LIN {X 0,Y 72.72,Z 376.859,A -85,B 0,C 180,E1 -30203.104,E2 -30203.104} C_VEL
LIN {X 0,Y 74.834,Z 373.573,A -85,B 0,C 180,E1 -30209.448,E2 -30209.448} C_VEL
LIN {X 0,Y 76.166,Z 370.91,A -85,B 0,C 180,E1 -30214.53,E2 -30214.53} C_VEL
LIN {X 0,Y 77.498,Z 367.967,A -85,B 0,C 180,E1 -30221.527,E2 -30221.527} C_VEL
LIN {X 0,Y 78.253,Z 365.544,A -85,B 0,C 180,E1 -30229.683,E2 -30229.683} C_VEL
LIN {X 0,Y 78.687,Z 364.699,A -85,B 0,C 180,E1 -30234.216,E2 -30234.216} C_VEL
LIN {X 0,Y 78.512,Z 364.725,A -85,B 0,C 180,E1 -30236.541,E2 -30236.541} C_VEL
LIN {X 0,Y 77.196,Z 365.763,A -85,B 0,C 180,E1 -30239.68,E2 -30239.68} C_VEL
LIN {X 0,Y 72.784,Z 369.848,A -85,B 0,C 180,E1 -30247.513,E2 -30247.513} C_VEL
LIN {X 0,Y 72.396,Z 370.336,A -85,B 0,C 180,E1 -30249.099,E2 -30249.099} C_VEL
LIN {X 0,Y 71.855,Z 371.227,A -85,B 0,C 180,E1 -30252.026,E2 -30252.026} C_VEL
LIN {X 0,Y 71.087,Z 372.22,A -85,B 0,C 180,E1 -30254.34,E2 -30254.34} C_VEL
LIN {X 0,Y 69.527,Z 373.648,A -85,B 0,C 180,E1 -30256.205,E2 -30256.205} C_VEL
LIN {X 0,Y 68.06,Z 374.817,A -85,B 0,C 180,E1 -30257.224,E2 -30257.224} C_VEL
LIN {X 0,Y 57.01,Z 381.349,A -85,B 0,C 180,E1 -30262.4,E2 -30262.4} C_VEL
LIN {X 0,Y 47.981,Z 385.676,A -85,B 0,C 180,E1 -30268.5,E2 -30268.5} C_VEL
LIN {X 0,Y 42.377,Z 388.048,A -85,B 0,C 180,E1 -30273.983,E2 -30273.983} C_VEL
LIN {X 0,Y 37.23,Z 389.851,A -85,B 0,C 180,E1 -30280.969,E2 -30280.969} C_VEL
LIN {X 0,Y 29.547,Z 392.319,A -85,B 0,C 180,E1 -30301.595,E2 -30301.595} C_VEL
LIN {X 0,Y 27.527,Z 392.919,A -85,B 0,C 180,E1 -30315.208,E2 -30315.208} C_VEL
LIN {X 0,Y 27.087,Z 393.084,A -85,B 0,C 180,E1 -30330,E2 -30330} C_VEL
LIN {X 0,Y 27.51,Z 392.918,A -85,B 0,C 180,E1 -30344.801,E2 -30344.801} C_VEL
LIN {X 0,Y 29.494,Z 392.317,A -85,B 0,C 180,E1 -30358.461,E2 -30358.461} C_VEL
LIN {X 0,Y 37.219,Z 389.851,A -85,B 0,C 180,E1 -30379.051,E2 -30379.051} C_VEL
LIN {X 0,Y 45.142,Z 386.896,A -85,B 0,C 180,E1 -30388.898,E2 -30388.898} C_VEL
LIN {X 0,Y 53.964,Z 382.905,A -85,B 0,C 180,E1 -30395.73,E2 -30395.73} C_VEL
LIN {X 0,Y 63.273,Z 377.774,A -85,B 0,C 180,E1 -30400.743,E2 -30400.743} C_VEL
LIN {X 0,Y 68.055,Z 374.817,A -85,B 0,C 180,E1 -30402.789,E2 -30402.789} C_VEL
LIN {X 0,Y 69.524,Z 373.648,A -85,B 0,C 180,E1 -30403.803,E2 -30403.803} C_VEL
LIN {X 0,Y 71.069,Z 372.231,A -85,B 0,C 180,E1 -30405.656,E2 -30405.656} C_VEL
LIN {X 0,Y 72.083,Z 370.933,A -85,B 0,C 180,E1 -30408.723,E2 -30408.723} C_VEL
LIN {X 0,Y 73.11,Z 369.368,A -85,B 0,C 180,E1 -30414.452,E2 -30414.452} C_VEL
LIN {X 0,Y 73.872,Z 368.359,A -85,B 0,C 180,E1 -30419.968,E2 -30419.968} C_VEL
LIN {X 0,Y 72.867,Z 369.184,A -85,B 0,C 180,E1 -30426.331,E2 -30426.331} C_VEL
LIN {X 0,Y 72.009,Z 370.387,A -85,B 0,C 180,E1 -30432.587,E2 -30432.587} C_VEL
LIN {X 0,Y 71.53,Z 371.492,A -85,B 0,C 180,E1 -30437.108,E2 -30437.108} C_VEL
LIN {X 0,Y 70.166,Z 373.929,A -85,B 0,C 180,E1 -30443.581,E2 -30443.581} C_VEL
LIN {X 0,Y 69.095,Z 375.402,A -85,B 0,C 180,E1 -30447.196,E2 -30447.196} C_VEL
LIN {X 0,Y 67.095,Z 378.1,A -85,B 0,C 180,E1 -30453.075,E2 -30453.075} C_VEL
LIN {X 0,Y 63.076,Z 382.804,A -85,B 0,C 180,E1 -30464.263,E2 -30464.263} C_VEL
LIN {X 0,Y 61.501,Z 386.014,A -85,B 0,C 180,E1 -30475.155,E2 -30475.155} C_VEL
LIN {X 0,Y 62.216,Z 387.991,A -85,B 0,C 180,E1 -30484.551,E2 -30484.551} C_VEL
LIN {X 0,Y 66.715,Z 389.818,A -85,B 0,C 180,E1 -30497.838,E2 -30497.838} C_VEL
LIN {X 0,Y 70.841,Z 390.257,A -85,B 0,C 180,E1 -30504.307,E2 -30504.307} C_VEL
LIN {X 0,Y 75.986,Z 390.258,A -85,B 0,C 180,E1 -30510,E2 -30510} C_VEL
LIN {X 0,Y 70.616,Z 390.238,A -85,B 0,C 180,E1 -30515.961,E2 -30515.961} C_VEL
LIN {X 0,Y 65.397,Z 389.543,A -85,B 0,C 180,E1 -30524.869,E2 -30524.869} C_VEL
LIN {X 0,Y 61.939,Z 387.669,A -85,B 0,C 180,E1 -30536.991,E2 -30536.991} C_VEL
LIN {X 0,Y 61.564,Z 385.453,A -85,B 0,C 180,E1 -30547.024,E2 -30547.024} C_VEL
LIN {X 0,Y 63.998,Z 381.588,A -85,B 0,C 180,E1 -30558.837,E2 -30558.837} C_VEL
LIN {X 0,Y 67.094,Z 378.1,A -85,B 0,C 180,E1 -30566.926,E2 -30566.926} C_VEL
LIN {X 0,Y 69.778,Z 374.487,A -85,B 0,C 180,E1 -30575.019,E2 -30575.019} C_VEL
LIN {X 0,Y 70.905,Z 372.605,A -85,B 0,C 180,E1 -30579.738,E2 -30579.738} C_VEL
LIN {X 0,Y 71.576,Z 371.46,A -85,B 0,C 180,E1 -30582.904,E2 -30582.904} C_VEL
LIN {X 0,Y 72.257,Z 370.036,A -85,B 0,C 180,E1 -30588.817,E2 -30588.817} C_VEL
LIN {X 0,Y 73.07,Z 368.988,A -85,B 0,C 180,E1 -30594.822,E2 -30594.822} C_VEL
LIN {X 0,Y 73.883,Z 368.35,A -85,B 0,C 180,E1 -30600.032,E2 -30600.032} C_VEL
LIN {X 0,Y 73.103,Z 369.373,A -85,B 0,C 180,E1 -30605.549,E2 -30605.549} C_VEL
LIN {X 0,Y 72.396,Z 370.336,A -85,B 0,C 180,E1 -30609.099,E2 -30609.099} C_VEL
LIN {X 0,Y 71.537,Z 371.196,A -85,B 0,C 180,E1 -30610.75,E2 -30610.75} C_VEL
LIN {X 0,Y 69.503,Z 372.798,A -85,B 0,C 180,E1 -30612.197,E2 -30612.197} C_VEL
LIN {X 0,Y 65.793,Z 375.28,A -85,B 0,C 180,E1 -30613.316,E2 -30613.316} C_VEL
LIN {X 0,Y 56.47,Z 380.309,A -85,B 0,C 180,E1 -30614.749,E2 -30614.749} C_VEL
LIN {X 0,Y 55.18,Z 380.901,A -85,B 0,C 180,E1 -30615.229,E2 -30615.229} C_VEL
LIN {X 0,Y 45.014,Z 385.481,A -85,B 0,C 180,E1 -30620.486,E2 -30620.486} C_VEL
LIN {X 0,Y 38.846,Z 387.852,A -85,B 0,C 180,E1 -30625.233,E2 -30625.233} C_VEL
LIN {X 0,Y 32.995,Z 389.656,A -85,B 0,C 180,E1 -30631.571,E2 -30631.571} C_VEL
LIN {X 0,Y 23.526,Z 392.123,A -85,B 0,C 180,E1 -30653.313,E2 -30653.313} C_VEL
LIN {X 0,Y 20.721,Z 392.724,A -85,B 0,C 180,E1 -30670.174,E2 -30670.174} C_VEL
LIN {X 0,Y 19.994,Z 392.889,A -85,B 0,C 180,E1 -30690,E2 -30690} C_VEL
LIN {X 0,Y 20.704,Z 392.723,A -85,B 0,C 180,E1 -30709.843,E2 -30709.843} C_VEL
LIN {X 0,Y 23.483,Z 392.122,A -85,B 0,C 180,E1 -30726.765,E2 -30726.765} C_VEL
LIN {X 0,Y 32.987,Z 389.655,A -85,B 0,C 180,E1 -30748.45,E2 -30748.45} C_VEL
LIN {X 0,Y 41.907,Z 386.701,A -85,B 0,C 180,E1 -30757.271,E2 -30757.271} C_VEL
LIN {X 0,Y 51.45,Z 382.71,A -85,B 0,C 180,E1 -30762.974,E2 -30762.974} C_VEL
LIN {X 0,Y 61.285,Z 377.577,A -85,B 0,C 180,E1 -30767.077,E2 -30767.077} C_VEL
LIN {X 0,Y 64.617,Z 375.658,A -85,B 0,C 180,E1 -30768.196,E2 -30768.196} C_VEL
LIN {X 0,Y 66.311,Z 374.202,A -85,B 0,C 180,E1 -30771.201,E2 -30771.201} C_VEL
LIN {X 0,Y 66.824,Z 373.516,A -85,B 0,C 180,E1 -30773.928,E2 -30773.928} C_VEL
LIN {X 0,Y 67.857,Z 372.402,A -85,B 0,C 180,E1 -30779.965,E2 -30779.965} C_VEL
LIN {X 0,Y 66.889,Z 373.083,A -85,B 0,C 180,E1 -30785.995,E2 -30785.995} C_VEL
LIN {X 0,Y 65.56,Z 374.822,A -85,B 0,C 180,E1 -30795.254,E2 -30795.254} C_VEL
LIN {X 0,Y 64.719,Z 375.828,A -85,B 0,C 180,E1 -30798.973,E2 -30798.973} C_VEL
LIN {X 0,Y 63.815,Z 376.916,A -85,B 0,C 180,E1 -30802.322,E2 -30802.322} C_VEL
LIN {X 0,Y 62.281,Z 378.666,A -85,B 0,C 180,E1 -30806.788,E2 -30806.788} C_VEL
LIN {X 0,Y 60.863,Z 380.042,A -85,B 0,C 180,E1 -30810.584,E2 -30810.584} C_VEL
LIN {X 0,Y 58.133,Z 382.586,A -85,B 0,C 180,E1 -30817.138,E2 -30817.138} C_VEL
LIN {X 0,Y 54.887,Z 386.242,A -85,B 0,C 180,E1 -30830.193,E2 -30830.193} C_VEL
LIN {X 0,Y 54.952,Z 388.627,A -85,B 0,C 180,E1 -30843.438,E2 -30843.438} C_VEL
LIN {X 0,Y 58.246,Z 390.056,A -85,B 0,C 180,E1 -30856.036,E2 -30856.036} C_VEL
LIN {X 0,Y 63.4,Z 390.596,A -85,B 0,C 180,E1 -30865.533,E2 -30865.533} C_VEL
LIN {X 0,Y 66.98,Z 390.505,A -85,B 0,C 180,E1 -30870,E2 -30870} C_VEL
LIN {X 0,Y 62.009,Z 390.5,A -85,B 0,C 180,E1 -30876.508,E2 -30876.508} C_VEL
LIN {X 0,Y 58.018,Z 390.03,A -85,B 0,C 180,E1 -30884.463,E2 -30884.463} C_VEL
LIN {X 0,Y 54.544,Z 387.901,A -85,B 0,C 180,E1 -30901.023,E2 -30901.023} C_VEL
LIN {X 0,Y 55.576,Z 385.162,A -85,B 0,C 180,E1 -30914.067,E2 -30914.067} C_VEL
LIN {X 0,Y 59.376,Z 381.386,A -85,B 0,C 180,E1 -30925.948,E2 -30925.948} C_VEL
LIN {X 0,Y 60.835,Z 380.056,A -85,B 0,C 180,E1 -30929.4,E2 -30929.4} C_VEL
LIN {X 0,Y 62.553,Z 378.352,A -85,B 0,C 180,E1 -30934,E2 -30934} C_VEL
LIN {X 0,Y 63.828,Z 376.908,A -85,B 0,C 180,E1 -30937.689,E2 -30937.689} C_VEL
LIN {X 0,Y 65.607,Z 374.817,A -85,B 0,C 180,E1 -30944.596,E2 -30944.596} C_VEL
LIN {X 0,Y 66.036,Z 374.179,A -85,B 0,C 180,E1 -30947.748,E2 -30947.748} C_VEL
LIN {X 0,Y 66.901,Z 373.074,A -85,B 0,C 180,E1 -30954.006,E2 -30954.006} C_VEL
LIN {X 0,Y 67.864,Z 372.398,A -85,B 0,C 180,E1 -30960.035,E2 -30960.035} C_VEL
LIN {X 0,Y 66.493,Z 373.942,A -85,B 0,C 180,E1 -30967.788,E2 -30967.788} C_VEL
LIN {X 0,Y 66.326,Z 374.193,A -85,B 0,C 180,E1 -30968.804,E2 -30968.804} C_VEL
LIN {X 0,Y 64.62,Z 375.658,A -85,B 0,C 180,E1 -30971.818,E2 -30971.818} C_VEL
LIN {X 0,Y 55.18,Z 380.901,A -85,B 0,C 180,E1 -30975.229,E2 -30975.229} C_VEL
LIN {X 0,Y 49.984,Z 383.337,A -85,B 0,C 180,E1 -30976.863,E2 -30976.863} C_VEL
LIN {X 0,Y 40.668,Z 386.599,A -85,B 0,C 180,E1 -30978.07,E2 -30978.07} C_VEL
LIN {X 0,Y 31.155,Z 389.202,A -85,B 0,C 180,E1 -30980.11,E2 -30980.11} C_VEL
LIN {X 0,Y 25.796,Z 390.382,A -85,B 0,C 180,E1 -30984.48,E2 -30984.48} C_VEL
LIN {X 0,Y 18.32,Z 391.928,A -85,B 0,C 180,E1 -30999.896,E2 -30999.896} C_VEL
LIN {X 0,Y 14.238,Z 392.529,A -85,B 0,C 180,E1 -31020.422,E2 -31020.422} C_VEL
LIN {X 0,Y 12.888,Z 392.695,A -85,B 0,C 180,E1 -31050,E2 -31050} C_VEL
LIN {X 0,Y 14.221,Z 392.528,A -85,B 0,C 180,E1 -31079.616,E2 -31079.616} C_VEL
LIN {X 0,Y 18.29,Z 391.927,A -85,B 0,C 180,E1 -31100.219,E2 -31100.219} C_VEL
LIN {X 0,Y 29.882,Z 389.46,A -85,B 0,C 180,E1 -31120.175,E2 -31120.175} C_VEL
LIN {X 0,Y 39.702,Z 386.505,A -85,B 0,C 180,E1 -31126.8,E2 -31126.8} C_VEL
LIN {X 0,Y 49.828,Z 382.514,A -85,B 0,C 180,E1 -31130.854,E2 -31130.854} C_VEL
LIN {X 0,Y 60.041,Z 377.409,A -85,B 0,C 180,E1 -31133.734,E2 -31133.734} C_VEL
LIN {X 0,Y 60.973,Z 376.683,A -85,B 0,C 180,E1 -31136.658,E2 -31136.658} C_VEL
LIN {X 0,Y 61.603,Z 376.189,A -85,B 0,C 180,E1 -31139.962,E2 -31139.962} C_VEL
LIN {X 0,Y 60.449,Z 376.841,A -85,B 0,C 180,E1 -31146.637,E2 -31146.637} C_VEL
LIN {X 0,Y 59.409,Z 377.901,A -85,B 0,C 180,E1 -31153.644,E2 -31153.644} C_VEL
LIN {X 0,Y 58.673,Z 378.644,A -85,B 0,C 180,E1 -31156.618,E2 -31156.618} C_VEL
LIN {X 0,Y 57.028,Z 380.047,A -85,B 0,C 180,E1 -31161.652,E2 -31161.652} C_VEL
LIN {X 0,Y 55.058,Z 381.619,A -85,B 0,C 180,E1 -31166.683,E2 -31166.683} C_VEL
LIN {X 0,Y 51.473,Z 384.24,A -85,B 0,C 180,E1 -31174.994,E2 -31174.994} C_VEL
LIN {X 0,Y 48.331,Z 386.922,A -85,B 0,C 180,E1 -31186.567,E2 -31186.567} C_VEL
LIN {X 0,Y 47.921,Z 389.377,A -85,B 0,C 180,E1 -31203.899,E2 -31203.899} C_VEL
LIN {X 0,Y 50.658,Z 390.407,A -85,B 0,C 180,E1 -31215.993,E2 -31215.993} C_VEL
LIN {X 0,Y 58.044,Z 390.75,A -85,B 0,C 180,E1 -31230,E2 -31230} C_VEL
LIN {X 0,Y 50.64,Z 390.414,A -85,B 0,C 180,E1 -31243.923,E2 -31243.923} C_VEL
LIN {X 0,Y 47.685,Z 389.191,A -85,B 0,C 180,E1 -31257.945,E2 -31257.945} C_VEL
LIN {X 0,Y 48.85,Z 386.468,A -85,B 0,C 180,E1 -31275.999,E2 -31275.999} C_VEL
LIN {X 0,Y 52.59,Z 383.486,A -85,B 0,C 180,E1 -31287.742,E2 -31287.742} C_VEL
LIN {X 0,Y 55.041,Z 381.62,A -85,B 0,C 180,E1 -31293.352,E2 -31293.352} C_VEL
LIN {X 0,Y 57.028,Z 380.047,A -85,B 0,C 180,E1 -31298.348,E2 -31298.348} C_VEL
LIN {X 0,Y 58.689,Z 378.643,A -85,B 0,C 180,E1 -31303.331,E2 -31303.331} C_VEL
LIN {X 0,Y 59.465,Z 377.87,A -85,B 0,C 180,E1 -31306.369,E2 -31306.369} C_VEL
LIN {X 0,Y 60.5,Z 376.814,A -85,B 0,C 180,E1 -31313.369,E2 -31313.369} C_VEL
LIN {X 0,Y 61.606,Z 376.188,A -85,B 0,C 180,E1 -31320.038,E2 -31320.038} C_VEL
LIN {X 0,Y 60.979,Z 376.676,A -85,B 0,C 180,E1 -31323.29,E2 -31323.29} C_VEL
LIN {X 0,Y 60.054,Z 377.401,A -85,B 0,C 180,E1 -31326.257,E2 -31326.257} C_VEL
LIN {X 0,Y 52.905,Z 381.104,A -85,B 0,C 180,E1 -31328.1,E2 -31328.1} C_VEL
LIN {X 0,Y 43.039,Z 385.285,A -85,B 0,C 180,E1 -31331.556,E2 -31331.556} C_VEL
LIN {X 0,Y 36.385,Z 387.657,A -85,B 0,C 180,E1 -31335.035,E2 -31335.035} C_VEL
LIN {X 0,Y 25.796,Z 390.382,A -85,B 0,C 180,E1 -31344.48,E2 -31344.48} C_VEL
LIN {X 0,Y 20.638,Z 391.444,A -85,B 0,C 180,E1 -31351.235,E2 -31351.235} C_VEL
LIN {X 0,Y 15.305,Z 392.149,A -85,B 0,C 180,E1 -31359.453,E2 -31359.453} C_VEL
LIN {X 0,Y 6.636,Z 392.648,A -85,B 0,C 180,E1 -31408.258,E2 -31408.258} C_VEL
LIN {X 0,Y 9.258,Z 392.277,A -85,B 0,C 180,E1 -31466.038,E2 -31466.038} C_VEL
LIN {X 0,Y 14.777,Z 391.731,A -85,B 0,C 180,E1 -31482.02,E2 -31482.02} C_VEL
LIN {X 0,Y 28.272,Z 389.265,A -85,B 0,C 180,E1 -31493.88,E2 -31493.88} C_VEL
LIN {X 0,Y 38.701,Z 386.31,A -85,B 0,C 180,E1 -31497.147,E2 -31497.147} C_VEL
LIN {X 0,Y 49.201,Z 382.319,A -85,B 0,C 180,E1 -31499.095,E2 -31499.095} C_VEL
LIN {X 0,Y 55.18,Z 379.646,A -85,B 0,C 180,E1 -31499.957,E2 -31499.957} C_VEL
LIN {X 0,Y 53.81,Z 380.279,A -85,B 0,C 180,E1 -31507.46,E2 -31507.46} C_VEL
LIN {X 0,Y 51.911,Z 381.566,A -85,B 0,C 180,E1 -31515.662,E2 -31515.662} C_VEL
LIN {X 0,Y 49.361,Z 383.306,A -85,B 0,C 180,E1 -31522.276,E2 -31522.276} C_VEL
LIN {X 0,Y 43.53,Z 386.694,A -85,B 0,C 180,E1 -31536.173,E2 -31536.173} C_VEL
LIN {X 0,Y 41.177,Z 388.357,A -85,B 0,C 180,E1 -31546.945,E2 -31546.945} C_VEL
LIN {X 0,Y 40.535,Z 389.729,A -85,B 0,C 180,E1 -31559.979,E2 -31559.979} C_VEL
LIN {X 0,Y 43.293,Z 390.788,A -85,B 0,C 180,E1 -31576.658,E2 -31576.658} C_VEL
LIN {X 0,Y 49.152,Z 390.994,A -85,B 0,C 180,E1 -31590.093,E2 -31590.093} C_VEL
LIN {X 0,Y 43.28,Z 390.793,A -85,B 0,C 180,E1 -31603.268,E2 -31603.268} C_VEL
LIN {X 0,Y 40.47,Z 389.61,A -85,B 0,C 180,E1 -31621.397,E2 -31621.397} C_VEL
LIN {X 0,Y 42.022,Z 387.611,A -85,B 0,C 180,E1 -31638.09,E2 -31638.09} C_VEL
LIN {X 0,Y 47.355,Z 384.384,A -85,B 0,C 180,E1 -31653.619,E2 -31653.619} C_VEL
LIN {X 0,Y 49.355,Z 383.307,A -85,B 0,C 180,E1 -31657.742,E2 -31657.742} C_VEL
LIN {X 0,Y 51.911,Z 381.566,A -85,B 0,C 180,E1 -31664.338,E2 -31664.338} C_VEL
LIN {X 0,Y 53.849,Z 380.261,A -85,B 0,C 180,E1 -31672.545,E2 -31672.545} C_VEL
LIN {X 0,Y 54.586,Z 379.927,A -85,B 0,C 180,E1 -31680.043,E2 -31680.043} C_VEL
LIN {X 0,Y 45.695,Z 383.849,A -85,B 0,C 180,E1 -31681.448,E2 -31681.448} C_VEL
LIN {X 0,Y 35.216,Z 387.462,A -85,B 0,C 180,E1 -31683.778,E2 -31683.778} C_VEL
LIN {X 0,Y 22.961,Z 390.346,A -85,B 0,C 180,E1 -31689.127,E2 -31689.127} C_VEL
LIN {X 0,Y 14.796,Z 391.733,A -85,B 0,C 180,E1 -31698.206,E2 -31698.206} C_VEL
LIN {X 0,Y 8.792,Z 392.334,A -85,B 0,C 180,E1 -31716.929,E2 -31716.929} C_VEL
LIN {X 0,Y 5.776,Z 392.5,A -85,B 0,C 180,E1 -31770,E2 -31770} C_VEL
LIN {X 0,Y 9.258,Z 392.277,A -85,B 0,C 180,E1 -31826.038,E2 -31826.038} C_VEL
LIN {X 0,Y 13.998,Z 391.792,A -85,B 0,C 180,E1 -31843.611,E2 -31843.611} C_VEL
LIN {X 0,Y 22.489,Z 390.364,A -85,B 0,C 180,E1 -31859.6,E2 -31859.6} C_VEL
LIN {X 0,Y 29.755,Z 388.809,A -85,B 0,C 180,E1 -31865.859,E2 -31865.859} C_VEL
LIN {X 0,Y 35.378,Z 387.289,A -85,B 0,C 180,E1 -31867.646,E2 -31867.646} C_VEL
LIN {X 0,Y 37.259,Z 386.682,A -85,B 0,C 180,E1 -31867.732,E2 -31867.732} C_VEL
LIN {X 0,Y 42.539,Z 384.895,A -85,B 0,C 180,E1 -31867.584,E2 -31867.584} C_VEL
LIN {X 0,Y 46.574,Z 383.48,A -85,B 0,C 180,E1 -31868.627,E2 -31868.627} C_VEL
LIN {X 0,Y 43.986,Z 384.706,A -85,B 0,C 180,E1 -31876.534,E2 -31876.534} C_VEL
LIN {X 0,Y 39.258,Z 386.918,A -85,B 0,C 180,E1 -31886.48,E2 -31886.48} C_VEL
LIN {X 0,Y 35.566,Z 388.585,A -85,B 0,C 180,E1 -31897.778,E2 -31897.778} C_VEL
LIN {X 0,Y 33.873,Z 390.761,A -85,B 0,C 180,E1 -31925.484,E2 -31925.484} C_VEL
LIN {X 0,Y 36.256,Z 391.214,A -85,B 0,C 180,E1 -31938.823,E2 -31938.823} C_VEL
LIN {X 0,Y 40.491,Z 391.231,A -85,B 0,C 180,E1 -31950,E2 -31950} C_VEL
LIN {X 0,Y 35.921,Z 391.175,A -85,B 0,C 180,E1 -31962.3,E2 -31962.3} C_VEL
LIN {X 0,Y 33.416,Z 390.281,A -85,B 0,C 180,E1 -31982.86,E2 -31982.86} C_VEL
LIN {X 0,Y 36.12,Z 388.289,A -85,B 0,C 180,E1 -32004.37,E2 -32004.37} C_VEL
LIN {X 0,Y 39.259,Z 386.918,A -85,B 0,C 180,E1 -32013.516,E2 -32013.516} C_VEL
LIN {X 0,Y 43.981,Z 384.706,A -85,B 0,C 180,E1 -32023.488,E2 -32023.488} C_VEL
LIN {X 0,Y 46.595,Z 383.471,A -85,B 0,C 180,E1 -32031.376,E2 -32031.376} C_VEL
LIN {X 0,Y 42.54,Z 384.895,A -85,B 0,C 180,E1 -32032.405,E2 -32032.405} C_VEL
LIN {X 0,Y 35.465,Z 387.267,A -85,B 0,C 180,E1 -32032.225,E2 -32032.225} C_VEL
LIN {X 0,Y 28.408,Z 389.07,A -85,B 0,C 180,E1 -32031.719,E2 -32031.719} C_VEL
LIN {X 0,Y 14.28,Z 391.537,A -85,B 0,C 180,E1 -32029.829,E2 -32029.829} C_VEL
LIN {X 0,Y 7.266,Z 392.139,A -85,B 0,C 180,E1 -32025.298,E2 -32025.298} C_VEL
LIN {X 0,Y 1.324,Z 392.305,A -85,B 0,C 180,E1 -31950,E2 -31950} C_VEL
LIN {X 0,Y 7.277,Z 392.137,A -85,B 0,C 180,E1 -31875.035,E2 -31875.035} C_VEL
LIN {X 0,Y 14.29,Z 391.535,A -85,B 0,C 180,E1 -31870.389,E2 -31870.389} C_VEL
LIN {X 0,Y 28.409,Z 389.07,A -85,B 0,C 180,E1 -31868.298,E2 -31868.298} C_VEL
LIN {X 0,Y 37.259,Z 386.682,A -85,B 0,C 180,E1 -31867.732,E2 -31867.732} C_VEL
LIN {X 0,Y 36.338,Z 387.038,A -85,B 0,C 180,E1 -31869.593,E2 -31869.593} C_VEL
LIN {X 0,Y 30.177,Z 388.702,A -85,B 0,C 180,E1 -31874.852,E2 -31874.852} C_VEL
LIN {X 0,Y 19.853,Z 390.891,A -85,B 0,C 180,E1 -31886.666,E2 -31886.666} C_VEL
LIN {X 0,Y 12.837,Z 391.838,A -85,B 0,C 180,E1 -31905.11,E2 -31905.11} C_VEL
LIN {X 0,Y 10.847,Z 391.963,A -85,B 0,C 180,E1 -31915.428,E2 -31915.428} C_VEL
LIN {X 0,Y 8.441,Z 392.11,A -85,B 0,C 180,E1 -31950,E2 -31950} C_VEL
LIN {X 0,Y 11.388,Z 391.943,A -85,B 0,C 180,E1 -31988.106,E2 -31988.106} C_VEL
LIN {X 0,Y 17.054,Z 391.341,A -85,B 0,C 180,E1 -32005.505,E2 -32005.505} C_VEL
LIN {X 0,Y 30.261,Z 388.875,A -85,B 0,C 180,E1 -32018.271,E2 -32018.271} C_VEL
LIN {X 0,Y 32.537,Z 388.342,A -85,B 0,C 180,E1 -32017.604,E2 -32017.604} C_VEL
LIN {X 0,Y 26.458,Z 390.817,A -85,B 0,C 180,E1 -31987.319,E2 -31987.319} C_VEL
LIN {X 0,Y 28.587,Z 391.54,A -85,B 0,C 180,E1 -31960.918,E2 -31960.918} C_VEL
LIN {X 0,Y 31.813,Z 391.469,A -85,B 0,C 180,E1 -31950,E2 -31950} C_VEL
LIN {X 0,Y 27.918,Z 391.448,A -85,B 0,C 180,E1 -31935.42,E2 -31935.42} C_VEL
LIN {X 0,Y 26.543,Z 390.797,A -85,B 0,C 180,E1 -31912.443,E2 -31912.443} C_VEL
LIN {X 0,Y 32.531,Z 388.344,A -85,B 0,C 180,E1 -31882.407,E2 -31882.407} C_VEL
LIN {X 0,Y 30.264,Z 388.875,A -85,B 0,C 180,E1 -31881.741,E2 -31881.741} C_VEL
LIN {X 0,Y 17.082,Z 391.34,A -85,B 0,C 180,E1 -31894.628,E2 -31894.628} C_VEL
LIN {X 0,Y 10.847,Z 391.963,A -85,B 0,C 180,E1 -31915.428,E2 -31915.428} C_VEL
LIN {X 0,Y 9.403,Z 392.092,A -85,B 0,C 180,E1 -31939.357,E2 -31939.357} C_VEL
LIN {X 0,Y 10.847,Z 392.071,A -85,B 0,C 180,E1 -31963.556,E2 -31963.556} C_VEL
LIN {X 0,Y 14.217,Z 391.907,A -85,B 0,C 180,E1 -31977.798,E2 -31977.798} C_VEL
LIN {X 0,Y 17.583,Z 391.639,A -85,B 0,C 180,E1 -31980.568,E2 -31980.568} C_VEL
LIN {X 0,Y 19.191,Z 391.552,A -85,B 0,C 180,E1 -31978.536,E2 -31978.536} C_VEL
LIN {X 0,Y 19.426,Z 391.563,A -85,B 0,C 180,E1 -31977.145,E2 -31977.145} C_VEL
LIN {X 0,Y 23.197,Z 391.705,A -85,B 0,C 180,E1 -31950,E2 -31950} C_VEL
LIN {X 0,Y 19.477,Z 391.56,A -85,B 0,C 180,E1 -31922.845,E2 -31922.845} C_VEL
LIN {X 0,Y 17.573,Z 391.748,A -85,B 0,C 180,E1 -31926.427,E2 -31926.427} C_VEL
LIN {X 0,Y 15.545,Z 391.915,A -85,B 0,C 180,E1 -31950,E2 -31950} C_VEL
LIN {X 0,Y 17.54,Z 391.749,A -85,B 0,C 180,E1 -31973.621,E2 -31973.621} C_VEL
LIN {X 0,Y 19.426,Z 391.563,A -85,B 0,C 180,E1 -31977.145,E2 -31977.145} C_VEL
LIN {X 0,Y 21.342,Z 393.556,A -85,B 0,C 180,E1 -31979.997,E2 -31979.997} C_VEL
LIN {X 0,Y 21.342,Z 600,A -85,B 0,C 180,E1 -31979.997,E2 -31979.997} C_VEL
LIN {X 0,Y 21.342,Z 600,A -85,B 0,C 180,E1 -31979.997,E2 -31979.997}

QRS_NEXT_CUT()

QRS_NEXT()
QRS_HOME()

END
